PROGRAM PG_Heizung
VAR
	FB_Heizung_0: FB_Heizung;
END_VAR

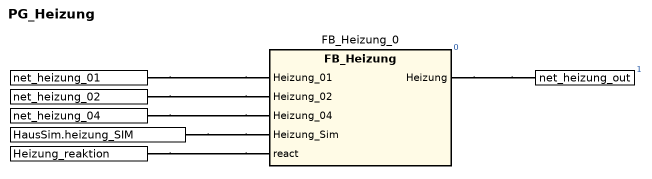
FB_Heizung_0(
    Heizung_01 := net_heizung_01,
    Heizung_02 := net_heizung_02,
    Heizung_04 := net_heizung_04,
    Heizung_Sim := HausSim.heizung_SIM,
    react := Heizung_reaktion); // FB_Heizung
net_heizung_out := FB_Heizung_0.Heizung;

END_PROGRAM

(* stored: Version 1.1.0.1, ProductVersion 3.1.4018.5
   POU PG_Heizung: Id {3b5956ba-ccdb-470d-8ac9-789b7ff9553e}, SpecialFunc None *)
